(* IEC 61131-3 sources: actuators/src, 7 files *)

(* ---- ActuatorState.st ---- *)
NAMESPACE Simatic.Ax.Actuators

    // Enumeration representing the possible states of an actuator.
    TYPE
        ActuatorState : (
            InHomePosition,       // 0: Actuator is in the home position.
            MoveToWorkPosition,   // 1: Actuator is moving to the first work position.
            MoveToWorkPosition2,  // 2: Actuator is moving to the second work position.
            InWorkPosition,       // 3: Actuator is in the first work position.
            InWorkPosition2,      // 4: Actuator is in the second work position.
            MoveToHomePosition,   // 5: Actuator is moving to the home position.
            Error,                // 6: Actuator is in an error state.
            Undefined             // 7: Actuator state is undefined.
        ) := Undefined;
    END_TYPE

END_NAMESPACE

(* ---- itfActuator.st ---- *)
USING Simatic.Ax.Commands;
USING Simatic.Ax.Commands;

NAMESPACE Simatic.Ax.Actuators

    // Interface for actuators, defining methods for controlling actuator states and retrieving their current state.
    INTERFACE itfActuator
        // Command to move the actuator to the home position.
        METHOD GoToHomePosition : itfCommand
        END_METHOD

        // Command to move the actuator to the first work position.
        METHOD GoToWorkPosition : itfCommand
        END_METHOD

        // Command to move the actuator to the second work position.
        METHOD GoToWorkPosition2 : itfCommand
        END_METHOD

        // Command to reset the actuator
        METHOD Reset
        END_METHOD

        // Retrieves the current state of the actuator.
        METHOD GetState : ActuatorState
        END_METHOD
    END_INTERFACE

END_NAMESPACE

(* ---- ToString.st ---- *)
NAMESPACE Simatic.Ax.Actuators

    FUNCTION INTERNAL ToString : STRING
        VAR_INPUT
            val : ActuatorState;
        END_VAR
        CASE val OF
            ActuatorState#InHomePosition:
                ToString := 'InHomePosition';
                RETURN;
            ActuatorState#MoveToWorkPosition:
                ToString := 'MoveToWorkPosition';
                RETURN;
            ActuatorState#MoveToWorkPosition2:
                ToString := 'MoveToWorkPosition2';
                RETURN;
            ActuatorState#InWorkPosition:
                ToString := 'InWorkPosition';
                RETURN;
            ActuatorState#InWorkPosition2:
                ToString := 'InWorkPosition2';
                RETURN;
            ActuatorState#MoveToHomePosition:
                ToString := 'MoveToHomePosition';
                RETURN;
            ActuatorState#Error:
                ToString := 'Error';
                RETURN;
            ActuatorState#Undefined:
                ToString := 'Undefined';
                RETURN;
        END_CASE;
        ;
    END_FUNCTION

END_NAMESPACE

(* ---- Actuator2Way.st ---- *)
NAMESPACE Simatic.Ax.Actuators

    // Represents a 2-way actuator that can move between two positions: Home and Work.
    CLASS Actuator2Way
        EXTENDS ActuatorBase
        VAR PUBLIC
        // Public variables can be declared here if needed.
        END_VAR

        // Initializes the actuator. This method is called during the setup phase.
        METHOD PROTECTED OVERRIDE InitActuator
            ;
        END_METHOD

        // Executes the actuator logic based on its current state and sensor inputs.
        METHOD PROTECTED OVERRIDE ExecuteActuator
            VAR_TEMP
                _isInHomePos, _isInWorkPos : BOOL; // Flags for sensor states.
                _currentState : ActuatorState;    // Current state of the actuator.
            END_VAR

            // Ensure the output to work position is not null.
            IF (Q_ToWorkPosition = NULL) THEN
                THIS.SetError(WORD#16#8101); // Set error code for invalid configuration.
                RETURN;
            END_IF;

            // Read sensor states.
            _isInHomePos := I_InHomePosition.IsActivated();
            _currentState := THIS.GetState();
            _isInWorkPos := I_InWorkPosition.IsActivated();

            // Handle state transitions based on the current state.
            CASE _currentState OF
                //##############################################
                // Undefined: Determine the actuator's position.
                //##############################################
                ActuatorState#Undefined:
                    IF NOT (_isInHomePos) AND NOT (_isInWorkPos) THEN
                        THIS.ChangeState(ActuatorState#MoveToHomePosition);
                    ELSIF (_isInHomePos) AND NOT (_isInWorkPos) THEN
                        THIS.ChangeState(ActuatorState#InHomePosition);
                    ELSIF NOT (_isInHomePos) AND (_isInWorkPos) THEN
                        THIS.ChangeState(ActuatorState#InWorkPosition);
                    ELSE
                        ; // Error: Both sensors are activated.
                    END_IF;

                //##############################################
                // InHomePosition: Hold the home position.
                //##############################################
                ActuatorState#InHomePosition:
                    THIS.SetDone();
                    Q_ToHomePosition.Hold();

                //##############################################
                // Move to Work position: Transition to work position.
                //##############################################
                ActuatorState#MoveToWorkPosition:
                    IF THIS.StateHasChanged() THEN
                        _toWorkPosCounter := _toWorkPosCounter + 1;
                        Q_ToWorkPosition.Set();
                        Q_ToHomePosition.Reset();
                        I_InHomePosition.EnableSupervision(Mode := SuperVisionMode#Action);
                        I_InWorkPosition.EnableSupervision(Mode := SuperVisionMode#Reaction);
                    END_IF;
                    IF (I_InWorkPosition.IsActivated()) THEN
                        I_InWorkPosition.EnableSupervision(Mode := SupervisionMode#PositionControl);
                        I_InHomePosition.EnableSupervision(Mode := SuperVisionMode#PositionControl);
                        THIS.SetDone();
                        Q_ToWorkPosition.Hold();
                        THIS.ChangeState(ActuatorState#InWorkPosition);
                    END_IF;

                //##############################################
                // InWorkPosition: Hold the work position.
                //##############################################
                ActuatorState#InWorkPosition:
                    THIS.SetDone();
                    Q_ToWorkPosition.Hold();

                //##############################################
                // Move to Home position: Transition to home position.
                //##############################################
                ActuatorState#MoveToHomePosition:
                    IF (THIS.StateHasChanged()) THEN
                        _toHomePosCounter := _toHomePosCounter + 1;
                        Q_ToHomePosition.Set();
                        Q_ToWorkPosition.Reset();
                        I_InWorkPosition.EnableSupervision(Mode := SuperVisionMode#Action);
                        I_InHomePosition.EnableSupervision(Mode := SuperVisionMode#Reaction);
                    END_IF;
                    IF (I_InHomePosition.IsActivated()) THEN
                        I_InHomePosition.EnableSupervision(Mode := SupervisionMode#PositionControl);
                        I_InWorkPosition.EnableSupervision(Mode := SuperVisionMode#PositionControl);
                        THIS.ChangeState(ActuatorState#InHomePosition);
                        Q_ToHomePosition.Hold();
                        THIS.SetDone();
                    END_IF;

                //##############################################
                // Error: Handle error state.
                //##############################################
                ActuatorState#Error:
                    _errorCounter := _errorCounter + 1;
                    Q_ToHomePosition.Reset();
                    Q_ToWorkPosition.Reset();

            END_CASE;
        END_METHOD

        METHOD PUBLIC OVERRIDE OnNotification
            // Read Error States of Endswitch
            _notificationCounter := _notificationCounter + 1;
            I_InHomePosition.GetError();
            I_InWorkPosition.GetError();
            THIS.SetError(WORD#16#8201);
            THIS.ChangeState(ActuatorState#Error);
        END_METHOD

    END_CLASS

END_NAMESPACE

(* ---- Actuator3Way.st ---- *)
USING Simatic.Ax.Commands;
USING System.Timer;

NAMESPACE Simatic.Ax.Actuators

    CLASS Actuator3Way
        EXTENDS ActuatorBase
        VAR PUBLIC
            I_InWorkPosition2 : itfEndswitch;
            Q_ToWorkPosition2 : itfPositionControl;
        END_VAR
        VAR PROTECTED
            _MonitoringTimer : System.Timer.OnDelay;
            _simFeedbackWorkPos2, _hasActiveToWork2 : BOOL;
            _ActualPosition : INT;
            _binSignalWorkPos2Null : NullEndswitch;
            _outSignalWhenNull : NullPositionControl;
        END_VAR

        METHOD PROTECTED OVERRIDE InitActuator
            IF (I_InWorkPosition2 = NULL) THEN
                I_InWorkPosition2 := _binSignalWorkPos2Null;
                _simFeedbackWorkPos2 := TRUE;
            END_IF;
            IF (Q_ToWorkPosition2 = NULL) THEN
                Q_ToWorkPosition2 := _outSignalWhenNull;
                _hasActiveToWork2 := FALSE;
            END_IF;
        END_METHOD

        METHOD PROTECTED OVERRIDE ExecuteActuator
            VAR_TEMP
                _isInHomePos, _isInWorkPos, _isInWorkPos2 : BOOL;
                _currentState : ActuatorState;
            END_VAR
            IF (Q_ToWorkPosition = NULL) THEN
                THIS.SetError(WORD#16#8101);
                RETURN;
            END_IF;
            _isInHomePos := I_InHomePosition.IsActivated();
            _isInWorkPos := I_InWorkPosition.IsActivated();
            _isInWorkPos2 := I_InWorkPosition2.IsActivated();
            _currentState := THIS.GetState();
            CASE _currentState OF
                //##############################################
                // Undefined
                //##############################################
                ActuatorState#Undefined:
                    // actuator is in between the two sensors (Home- and WorkPos)
                    IF NOT (_isInHomePos) AND NOT (_isInWorkPos) AND NOT (_isInWorkPos2) THEN
                        THIS.ChangeState(ActuatorState#MoveToHomePosition);
                    // actuator is in HomePos
                    ELSIF (_isInHomePos) AND NOT (_isInWorkPos) AND NOT (_isInWorkPos2) THEN
                        THIS.ChangeState(ActuatorState#InHomePosition);
                    // actuator is in any Workpos
                    ELSIF NOT (_isInHomePos) AND (_isInWorkPos OR _isInWorkPos2) THEN
                        THIS.ChangeState(ActuatorState#InWorkPosition);
                    // both sensors are activated --> undefined state
                    ELSE
                        ; // Error
                    END_IF;
                //##############################################
                // InHomePosition
                //##############################################
                ActuatorState#InHomePosition:
                    Q_ToHomePosition.Hold();
                    THIS.SetDone();
                // Received the command GoToWorkPosition switch on ToWorkPosition
                //##############################################
                // MoveToWorkPosition
                //##############################################
                ActuatorState#MoveToWorkPosition:
                    IF (I_InWorkPosition.IsActivated()) THEN
                        Q_ToWorkPosition.Hold();
                        THIS.SetDone();
                        THIS.ChangeState(ActuatorState#InWorkPosition);
                    END_IF;
                    IF (THIS.StateHasChanged()) THEN
                        Q_ToHomePosition.Reset();
                        Q_ToWorkPosition.Set();
                        Q_ToWorkPosition2.Reset();
                        I_InHomePosition.DisableMonitoring();
                        I_InWorkPosition2.DisableMonitoring();
                        I_InWorkPosition.StartMonitoring();
                    END_IF;
                //##############################################
                // InWorkPosition
                //##############################################
                // ### Actuator is in Workposition 1
                ActuatorState#InWorkPosition:
                    Q_ToWorkPosition.Hold();
                    THIS.SetDone();
                //##############################################
                // MoveToWorkPosition
                //##############################################
                ActuatorState#MoveToWorkPosition2:
                    IF (I_InWorkPosition2.IsActivated()) THEN
                        Q_ToWorkPosition2.Hold();
                        THIS.SetDone();
                        THIS.ChangeState(ActuatorState#InWorkPosition2);
                    END_IF;
                    IF (THIS.StateHasChanged()) THEN
                        Q_ToHomePosition.Reset();
                        Q_ToWorkPosition.Reset();
                        Q_ToWorkPosition2.Set();
                        I_InHomePosition.DisableMonitoring();
                        I_InWorkPosition.DisableMonitoring();
                        I_InWorkPosition2.StartMonitoring();
                    END_IF;
                //##############################################
                // InWorkPosition2
                //##############################################
                // ### Actuator is in Workposition 2
                ActuatorState#InWorkPosition2:
                    Q_ToWorkPosition2.Hold();
                    THIS.SetDone();
                //##############################################
                // Move to home position
                //##############################################
                ActuatorState#MoveToHomePosition:
                    IF (I_InHomePosition.IsActivated()) THEN
                        Q_ToHomePosition.Hold();
                        THIS.SetDone();
                        THIS.ChangeState(ActuatorState#InHomePosition);
                    END_IF;
                    IF (THIS.StateHasChanged()) THEN
                        Q_ToHomePosition.Set();
                        Q_ToWorkPosition.Reset();
                        Q_ToWorkPosition2.Reset();
                        I_InWorkPosition.DisableMonitoring();
                        I_InWorkPosition2.DisableMonitoring();
                        I_InHomePosition.StartMonitoring();
                    END_IF;
                ActuatorState#Error:
                    ;
            END_CASE;
        END_METHOD

        METHOD PUBLIC OVERRIDE GoToWorkPosition2 : itfCommand
            THIS.InitState();
            IF (I_InWorkPosition2 = NULL) THEN
                THIS.InitActuator();
            END_IF;
            IF (I_InWorkPosition2.IsActivated()) THEN
                THIS.ChangeState(ActuatorState#InWorkPosition2);
            ELSE
                THIS.ChangeState(ActuatorState#MoveToWorkPosition2);
            END_IF;
            GoToWorkPosition2 := THIS;
        END_METHOD
    END_CLASS

END_NAMESPACE

(* ---- ActuatorBase.st ---- *)
USING Simatic.Ax.AutomationFramework;
USING Simatic.Ax.Commands;
USING Simatic.Ax.AutomationFramework;

NAMESPACE Simatic.Ax.Actuators

    // Abstract base class for actuators, providing common functionality for actuator control.
    CLASS ABSTRACT ActuatorBase
        EXTENDS ExecuteControlModuleAbstract
        IMPLEMENTS itfActuator

        // Public variables
        VAR PUBLIC
            I_InHomePosition : itfEndswitch; // End switch indicating the actuator is in the home position.
            I_InWorkPosition : itfEndswitch; // End switch indicating the actuator is in the work position.
            Q_ToHomePosition : itfPositionControl;  // Command to move the actuator to the home position.
            Q_ToWorkPosition : itfPositionControl;  // Command to move the actuator to the work position.
            TimeToWork : LTIME := T#5s;
            TimeToHome : LTIME := T#5s;
        END_VAR

        VAR PROTECTED
            _toHomePosCounter : DINT;
            _toWorkPoscounter : DINT;
            _errorCounter : DINT;
            _notificationCounter : DINT;
        END_VAR

        // Private variables
        VAR PRIVATE
            _stateOld : ActuatorState;
            _currentState : ActuatorState;
            _stateHasChanged : BOOL;
            _simFeedbackHomePos : BOOL;
            _simFeedbackWorkPos : BOOL;
            _hasActiveToHome : BOOL := TRUE;
            _hasActiveToWork : BOOL := TRUE;
            _binSignalWorkPosNull : NullEndswitch;
            _binSignalHomePosNull : NullEndswitch;
            _outSignalWhenNull : NullPositionControl;
        END_VAR

        // Executes type-specific logic for the actuator.
        METHOD PROTECTED OVERRIDE _executeTypeSpecific
            _stateHasChanged := _currentState <> _stateOld;
            _stateOld := _currentState;
            IF (_simFeedbackHomePos) THEN
                _binSignalHomePosNull.ReadCyclic();
                ;
            END_IF;
            IF (_simFeedbackWorkPos) THEN
                _binSignalWorkPosNull.ReadCyclic();
                ;
            END_IF;
            THIS.ExecuteActuator();
        END_METHOD

        // Initializes the actuator's configuration.
        METHOD PROTECTED OVERRIDE _initmethod
            IF (I_InHomePosition = NULL) THEN
                I_InHomePosition := _binSignalHomePosNull;
                _binSignalHomePosNull.MonitoringTime := TimeToHome;
                _binSignalWorkPosNull.MonitoringTime := TimeToWork;
                _simFeedbackHomePos := TRUE;
            END_IF;
            IF (I_InWorkPosition = NULL) THEN
                I_InWorkPosition := _binSignalWorkPosNull;
                _simFeedbackWorkPos := TRUE;
            END_IF;
            IF (Q_ToWorkPosition = NULL) THEN
                Q_ToWorkPosition := _outSignalWhenNull;
                _hasActiveToWork := FALSE;
            END_IF;
            IF (Q_ToHomePosition = NULL) THEN
                Q_ToHomePosition := _outSignalWhenNull;
                _hasActiveToHome := FALSE;
            END_IF;
            THIS.InitActuator();
            ;
        END_METHOD

        // Executes actuator-specific logic. This method must be implemented by derived classes.
        METHOD PROTECTED ABSTRACT ExecuteActuator
        END_METHOD

        // Initializes the actuator. This method must be implemented by derived classes.
        METHOD PROTECTED ABSTRACT InitActuator
        END_METHOD

        // Retrieves the current state of the actuator.
        METHOD PUBLIC GetState : ActuatorState
            GetState := _currentState;
        END_METHOD

        // Command to move the actuator to the home position.
        METHOD PUBLIC GoToHomePosition : itfCommand
            THIS.InitState();
            IF (I_InHomePosition = NULL) THEN
                THIS._initmethod();
            END_IF;
            IF (I_InHomePosition.HasReached()) THEN
                _currentState := ActuatorState#InHomePosition;
            ELSE
                _currentState := ActuatorState#MoveToHomePosition;
            END_IF;
            GoToHomePosition := THIS;
            ;
        END_METHOD

        // Command to move the actuator to the first work position.
        METHOD PUBLIC GoToWorkPosition : itfCommand
            THIS.InitState();
            IF (I_InWorkPosition = NULL) THEN
                THIS._initmethod();
            END_IF;
            IF (I_InWorkPosition.IsActivated()) THEN
                _currentState := ActuatorState#InWorkPosition;
            ELSE
                _currentState := ActuatorState#MoveToWorkPosition;
            END_IF;
            GoToWorkPosition := THIS;
        END_METHOD

        // Command to move the actuator to the second work position.
        METHOD PUBLIC GoToWorkPosition2 : itfCommand
            THIS.SetDone();
            GoToWorkPosition2 := NULL;
        END_METHOD

        // Checks if the actuator's state has changed.
        METHOD PROTECTED StateHasChanged : BOOL
            StateHasChanged := _stateHasChanged;
        END_METHOD

        // Changes the current state of the actuator.
        METHOD PROTECTED ChangeState
            VAR_INPUT
                NewState : ActuatorState; // The new state to set for the actuator.
            END_VAR
            _currentState := NewState;
        END_METHOD

    END_CLASS

END_NAMESPACE

(* ---- TimeBasedActuator.st ---- *)
USING Simatic.Ax.Commands;
USING System.Timer;
USING Simatic.Ax.AutomationFramework;

NAMESPACE Simatic.Ax.Actuators
    CLASS TimeBasedActuator
        EXTENDS ActuatorBase
        VAR PUBLIC
            OnDuration : TIME;
        END_VAR
        VAR
            _tonOffDuration : OffDelay;
        END_VAR

        METHOD PROTECTED OVERRIDE InitActuator
            ;
        END_METHOD

        METHOD PROTECTED OVERRIDE ExecuteActuator
            VAR_TEMP
                _currentState : ActuatorState;
            END_VAR

            IF (Q_ToWorkPosition = NULL) THEN
                THIS.SetError(WORD#16#8101);
                RETURN;
            END_IF;
            _currentState := THIS.GetState();
            CASE _currentState OF
                // If undefined, go initial state:
                ActuatorState#Undefined:
                    THIS.ChangeState(ActuatorState#InHomePosition);
                // Switch all outputs off, when actuator is idle in home position
                ActuatorState#InHomePosition:
                    Q_ToWorkPosition.Reset();
                // Received the command GoToWorkPosition switch on ToWorkPosition
                ActuatorState#MoveToWorkPosition:
                    Q_ToWorkPosition.Set();
                    THIS.ChangeState(ActuatorState#InWorkPosition);
                // After Timeout switch off "ToWorkPosition"
                ActuatorState#InWorkPosition:
                    _tonOffDuration(signal := TRUE, Duration := OnDuration);
                    IF (_tonOffDuration.output) THEN
                        _tonOffDuration(signal := FALSE);
                        THIS.ChangeState(ActuatorState#MoveToHomePosition);
                        Q_ToWorkPosition.Reset();
                    END_IF;
                // Send done
                ActuatorState#MoveToHomePosition:
                    Q_ToWorkPosition.Reset();
                    THIS.ChangeState(ActuatorState#InHomePosition);
                    THIS.SetDone();
            END_CASE;
        END_METHOD

    END_CLASS

END_NAMESPACE
